FUNCTION_BLOCK DisposableCollection
VAR
	disposables : Stack;
END_VAR

METHOD PUBLIC DisposeAndRemoveAll
VAR
	disposable : I_Disposable;
END_VAR
WHILE disposables.TryPop(disposable) DO
	disposable.Dispose();
END_WHILE
END_METHOD

METHOD PUBLIC Insert
VAR_INPUT
	DisposableToInsert : I_Disposable;
END_VAR
disposables.Push(DisposableToInsert);
END_METHOD

END_FUNCTION_BLOCK

(* stored: Version 1.1.0.1, ProductVersion 3.1.4024.12
   POU DisposableCollection: Id {9e36cdcd-88ef-0310-24de-60899e6124c7}, SpecialFunc None
   Method DisposeAndRemoveAll: Id {318a25c1-4b89-0c0c-1ef1-19f5407dc5ec}
   Method Insert: Id {4ccca891-6202-09f4-1725-910f5f09648c} *)
